Yaskawa INFORM job: HOME.JBI

/JOB
//NAME HOME
//POS
///NPOS 1,1,0,0,0,0
///TOOL 0
///POSTYPE ROBOT
///RECTAN
///RCONF 0,0,0,0,0,0,0,0,0,0,0,0,0,0,0,0,0,0,0,0,0,0,0,0
C00000=1189.393,105.917,-803.391,44.6385,-7.3085,-43.6297
BC00000=1137.387,4350.236,1999.673
//INST
///DATE 2023/12/06 13:01
///ATTR SC,RW,RJ
////FRAME ROBOT
///GROUP1 RB1,BS1
NOP
MOVJ C00000 BC00000 VJ=20.00
END
